RoboDK station: RB KUKA.rdk

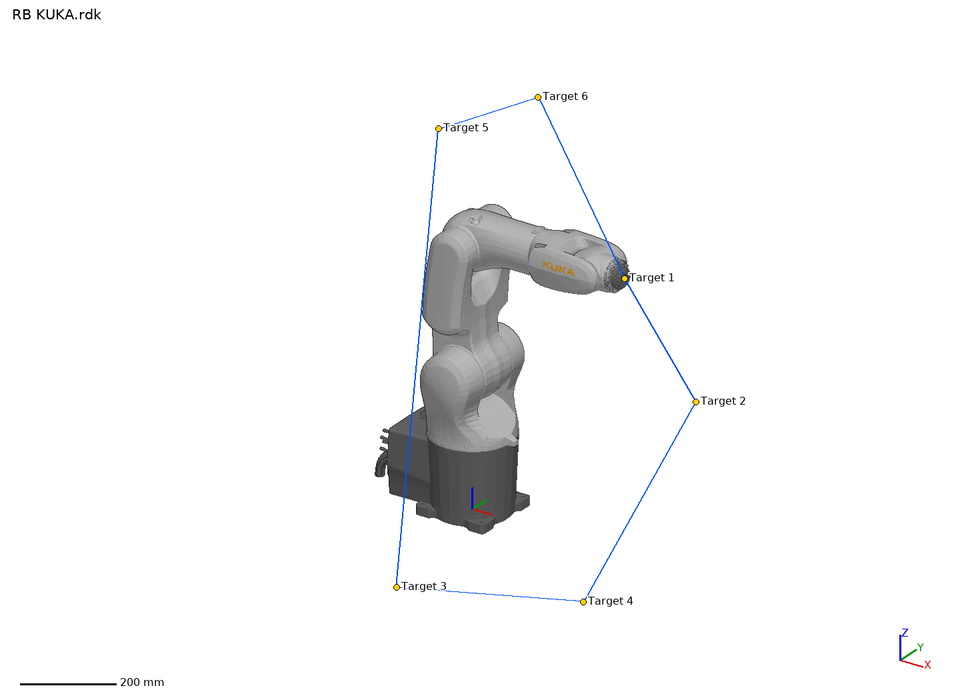
[picture v0: the station drawn from its stored meshes, robots at their saved joint values, targets as dots, program paths as lines]
Station New Station (2) (saved by RoboDK 5.5.4). Poses are relative to the parent item; angles as X-Y-Z fixed-axis rotations.
  - frame KUKA KR 4 R600 Base at (0, 0, 0) mm
    - robot KUKA KR 4 R600: 6 axes, payload 4.63 kg, reach 601 mm, repeatability 0.015 mm, weight 24 kg
        modified DH rows (alpha deg, a mm, theta deg, d mm): 0, 0, 0, 330; -90, 0, 0, 0; 0, 290, -90, 0; -90, 20, 0, 310; 90, 0, 0, 0; -90, 0, 180, 75
        joint limits [-170, -195, -115, -185, -120, -350] to [170, 40, 150, 180, 120, 350]; home [0, -90, 90, 0, 0, 0]; saved at [0, -90, 90, 0, 0, 0]
    - target Target 1 (Cartesian target) at (385, 0, 640) mm, rotated rx 0 ry 90 rz 0 deg; joints [0, -90, 90, 0, 0, 0] of KUKA KR 4 R600
    - target Target 2 (joint target) at (565.36, 0, 405.38) mm, rotated rx -179.46 ry 12.78 rz 2.44 deg; joints [0, -14.897, 4.813, 0, 112.872, -177.617] of KUKA KR 4 R600
    - target Target 4 (joint target) at (390.32, -155.98, -42.57) mm, rotated rx -176.2 ry 68.9 rz -16.43 deg; joints [21.6, 32.2, 9.454, 1.146, 117.284, -177.617] of KUKA KR 4 R600
    - target Target 3 (joint target) at (146.61, -484.66, 53.44) mm, rotated rx 16.15 ry 16.51 rz -82.96 deg; joints [70.359, 32.2, 9.454, 158.136, 117.284, -177.617] of KUKA KR 4 R600
    - target Target 5 (joint target) at (13.46, -142.51, 938.13) mm, rotated rx 17.87 ry -55.12 rz -69.4 deg; joints [73.625, -70.202, 2.479, 158.136, 77.464, -177.617] of KUKA KR 4 R600
    - target Target 6 (joint target) at (97.47, 98.01, 938.6) mm, rotated rx 6.03 ry -80.92 rz -130.73 deg; joints [146.219, -95.202, 1.432, 158.136, 77.464, -177.617] of KUKA KR 4 R600
  - program Prog1 (8 instructions, listed below)
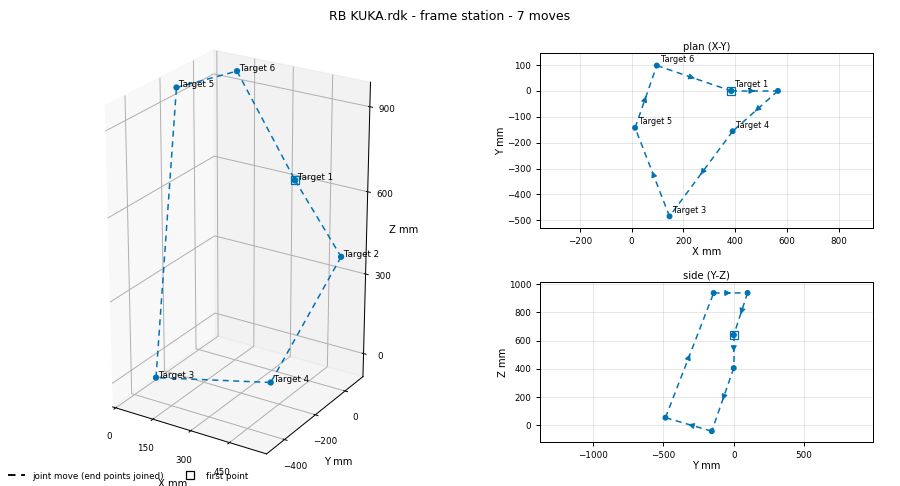
[picture p0: tool path of RB KUKA.rdk in frame station, 7 of 7 moves have a stored position in this frame; points joined in program order, loops and branches not executed]

--- program Prog1 (robot KUKA KR 4 R600) ---
  Set Ref.: KUKA KR 4 R600 Base
  MoveJ (Target 1)
  MoveJ (Target 2)
  MoveJ (Target 4)
  MoveJ (Target 3)
  MoveJ (Target 5)
  MoveJ (Target 6)
  MoveJ (Target 1)
